{attribute 'qualified_only'}
{attribute 'strict'}
TYPE eMode :
(
	MODE_MANUAL := 0,
	MODE_SINGLE := 1,
	MODE_AUTO := 2,
	MODE_MAINTENANCE := 3
);
END_TYPE

(* stored: Version 1.1.0.1, ProductVersion 3.1.4024.13
   DUT eMode: Id {3e645566-fce2-4812-9f11-298ed30b870b} *)
